FUNCTION_BLOCK PUBLIC FB_ModeVisualization IMPLEMENTS I_Mode
VAR_INPUT
END_VAR
VAR_OUTPUT
END_VAR
VAR
END_VAR

METHOD Auto
VAR_INPUT
	bEnable	: BOOL;
END_VAR
IF bEnable THEN
HMI.fCylinderPosition := CraneSimulation.fPositionAutoMode;
HMI.eMode := E_Mode.Auto; 
END_IF
END_METHOD

METHOD Manual
VAR_INPUT
	bEnable	: BOOL;
END_VAR
IF bEnable THEN
HMI.fCylinderPosition := HMI.fManualCylinderPositionReference;
HMI.eMode := E_Mode.Manual; 
END_IF
END_METHOD

METHOD Off
VAR_INPUT
	bEnable	: BOOL;
END_VAR
IF bEnable THEN
HMI.fCylinderPosition := 0;
HMI.eMode := E_Mode.Off; 
END_IF
END_METHOD

END_FUNCTION_BLOCK

(* stored: Version 1.1.0.1, ProductVersion 3.1.4024.10
   POU FB_ModeVisualization: Id {aba72860-427f-470a-b1b3-598fcfedf8ac}, SpecialFunc None
   Method Auto: Id {442e6fe3-95a7-4986-95ba-a5445c158c12}
   Method Manual: Id {35b2c634-f3ec-4586-a759-6cb663b58e39}
   Method Off: Id {8268ac46-d200-462b-ac0d-8adeeabf5eba} *)
